{attribute 'c++_compatible'}
FUNCTION_BLOCK MQTTClient_RobotState EXTENDS FB_IotMqttClient
VAR_INPUT
	{attribute 'TcEncoding':='UTF-8'}
	 sTopicRcv   : STRING(255);
	 {attribute 'TcEncoding':='UTF-8'}
	 sPayloadRcv : RobotState;
END_VAR
VAR_OUTPUT
END_VAR
VAR
END_VAR

{attribute 'c++_compatible'}
{attribute 'pack_mode' := '4'}
{attribute 'show'}
{attribute 'minimal_input_size' := '4'}
METHOD OnMqttMessage : HRESULT
VAR_IN_OUT CONSTANT
    topic    : STRING;
END_VAR
VAR_INPUT
    payload  : PVOID;
    length   : UDINT;
    qos      : TcIotMqttQos;
    repeated : BOOL;
END_VAR
VAR
    nPayloadRcvLen : UDINT;
END_VAR
STRNCPY( ADR(sTopicRcv), ADR(topic), SIZEOF(sTopicRcv) );
nPayloadRcvLen := MIN(length, DINT_TO_UDINT(SIZEOF(sPayloadRcv)));
MEMCPY( ADR(sPayloadRcv), payload, nPayloadRcvLen );

OnMqttMessage := S_OK;
END_METHOD

END_FUNCTION_BLOCK

(* stored: Version 1.1.0.1, ProductVersion 3.1.4024.10
   POU MQTTClient_RobotState: Id {21aef3f5-a9fe-4289-a0b1-2ce8601176b8}, SpecialFunc None
   Method OnMqttMessage: Id {0f1d807f-4524-456a-a0a6-71039b74cf06} *)
